// TIA Portal V17 export
// export: Created 2026-04-13T11:12:04.1208621Z, ExportSetting WithDefaults, DisplayName Totally Integrated Automation Portal, DisplayVersion V17 Update 4, DisplayName TIA Portal Openness, DisplayVersion V17 Update 4, DisplayName TIA Portal Version Control Interface, DisplayVersion V17, DisplayName SINAMICS Startdrive Advanced, DisplayVersion V17, DisplayName SINAMICS Startdrive G130, G150, S120, S150, SINAMICS MV, S210, DisplayVersion V17, DisplayName SINAMICS Startdrive G110M, G120, G120C, G120D, G120P, G115D, DisplayVersion V17, DisplayName STEP 7 Professional, DisplayVersion V17 Update 4, DisplayName STEP 7 Safety, DisplayVersion V17, DisplayName WinCC Professional, DisplayVersion V17 Update 4
FUNCTION_BLOCK "A5-模拟量输出"   // FB29, SCL
{ S7_Optimized_Access := 'TRUE' }
VERSION : 0.1
// stored: AutoNumber true, IsIECCheckEnabled false, IsRetainMemResEnabled false, MemoryReserve 100, SetENOAutomatically false, UDAEnableTagReadback false
   VAR
      进风加热比例调节阀 { S7_SetPoint := 'True'} : "A2-数据转换RTI";
      回风加热比例调节阀 { S7_SetPoint := 'True'} : "A2-数据转换RTI";
      放空比例调节阀 { S7_SetPoint := 'True'} : "A2-数据转换RTI";
   END_VAR
BEGIN
   REGION 模拟量输出
       #进风加热比例调节阀(I_Max := 27648,
                  I_Min := 5530,
                  R_Max := 100.0,
                  R_Min := 0.0,
                  R_Value := "SV".JF进风加热比例调节阀,
                  I_ChValue => "QWJF进风加热比例调节阀");

       #回风加热比例调节阀(I_Max := 27648,
                  I_Min := 5530,
                  R_Max := 100.0,
                  R_Min := 0.0,
                  R_Value := "SV".HF回风加热比例调节阀,
                  I_ChValue => "QWHF回风加热比例调节阀");

       #放空比例调节阀(I_Max := 27648,
                I_Min := 5530,
                R_Max := 100.0,
                R_Min := 0.0,
                R_Value := "SV".FK放空比例调节阀,
                I_ChValue => "QWFK放空比例调节阀");
   END_REGION
END_FUNCTION_BLOCK
